(* CoDeSys 2.3 export: ONOFF.EXP *)

(* POU Components/OnOff, ST *)
FUNCTION_BLOCK OnOff

VAR_INPUT
	input:BOOL;
END_VAR

VAR_OUTPUT
	output:BOOL;
END_VAR

VAR
	state:BOOL;
	EdgeDetection:EdgeDetection;
	tmp:BOOL;
END_VAR
EdgeDetection(input:=input, output => tmp);

IF tmp THEN
	state := NOT state;
END_IF

output := state;
END_FUNCTION_BLOCK
